(* IEC 61131-3 sources: ATCMcontrol_Engineering/src/Target/ATHW119/Libs/ATCM_IEC1131_3/table_23, 11 files *)

(* ---- ABS.st ---- *)
FUNCTION ABS : any_num
VAR_INPUT
    IN : any_num;
END_VAR

overload lreal(lreal)
inline
{
	%1
	abs_lreal
}

overload real(real)
inline
{
	%1
	abs_real
}

overload dint(dint)
inline
{
	%1
	abs_dint
}

overload int(int)
inline
{
	%1
	abs_int
}

END_FUNCTION

(* ---- ACOS.st ---- *)
FUNCTION ACOS : any_real
VAR_INPUT
    IN : any_real;
END_VAR

overload lreal(lreal) inline { STDLIB(acos_lreal) }
overload real(real)   inline { STDLIB(acos_real) }

END_FUNCTION

(* ---- ASIN.st ---- *)
FUNCTION ASIN : any_real
VAR_INPUT
    IN : any_real;
END_VAR

overload lreal(lreal) inline { STDLIB(asin_lreal) }
overload real(real) inline   { STDLIB(asin_real) }

END_FUNCTION

(* ---- ATAN.st ---- *)
FUNCTION ATAN : any_real
VAR_INPUT
    IN : any_real;
END_VAR

overload lreal(lreal) inline { STDLIB(atan_lreal) }
overload real(real)   inline { STDLIB(atan_real) }

END_FUNCTION

(* ---- COS.st ---- *)
FUNCTION COS : any_real
VAR_INPUT
    IN : any_real;
END_VAR

overload lreal(lreal) inline { STDLIB(cos_lreal) }
overload real(real) inline   { STDLIB(cos_real) }

END_FUNCTION

(* ---- EXP.st ---- *)
FUNCTION EXP : any_real
VAR_INPUT
    IN : any_real;
END_VAR

overload lreal(lreal) inline { STDLIB(exp_lreal) }
overload real(real)   inline { STDLIB(exp_real) }

END_FUNCTION

(* ---- LN.st ---- *)
FUNCTION LN : any_real
VAR_INPUT
    IN : any_real;
END_VAR

overload lreal(lreal) inline { STDLIB(log_lreal) }
overload real(real)   inline { STDLIB(log_real) }

END_FUNCTION

(* ---- LOG.st ---- *)
FUNCTION LOG : any_real
VAR_INPUT
    IN : any_real;
END_VAR

overload lreal(lreal) inline { STDLIB(log10_lreal) }
overload real(real)   inline { STDLIB(log10_real) }

END_FUNCTION

(* ---- SIN.st ---- *)
FUNCTION SIN : any_real
VAR_INPUT
    IN : any_real;
END_VAR

overload lreal(lreal) inline { STDLIB(sin_lreal) }
overload real(real)   inline { STDLIB(sin_real) }

END_FUNCTION

(* ---- sqrt.st ---- *)
FUNCTION SQRT : any_real
VAR_INPUT
    IN : any_real;
END_VAR

overload lreal(lreal) inline { STDLIB(sqrt_lreal) }
overload real(real) inline   { STDLIB(sqrt_real) }

END_FUNCTION

(* ---- TAN.st ---- *)
FUNCTION TAN : any_real
VAR_INPUT
    IN : any_real;
END_VAR

overload lreal(lreal) inline { STDLIB(tan_lreal) }
overload real(real)   inline { STDLIB(tan_real) }

END_FUNCTION
